# EPICS autosave request: xx_auto_transform_settings.req
$(P)$(T).DESC
$(P)$(T).SCAN
$(P)$(T).PREC
$(P)$(T).A
$(P)$(T).B
$(P)$(T).C
$(P)$(T).D
$(P)$(T).E
$(P)$(T).F
$(P)$(T).G
$(P)$(T).H
$(P)$(T).I
$(P)$(T).J
$(P)$(T).K
$(P)$(T).L
$(P)$(T).M
$(P)$(T).N
$(P)$(T).O
$(P)$(T).P
$(P)$(T).CMTA
$(P)$(T).CMTB
$(P)$(T).CMTC
$(P)$(T).CMTD
$(P)$(T).CMTE
$(P)$(T).CMTF
$(P)$(T).CMTG
$(P)$(T).CMTH
$(P)$(T).CMTI
$(P)$(T).CMTJ
$(P)$(T).CMTK
$(P)$(T).CMTL
$(P)$(T).CMTM
$(P)$(T).CMTN
$(P)$(T).CMTO
$(P)$(T).CMTP
$(P)$(T).CLCA
$(P)$(T).CLCB
$(P)$(T).CLCC
$(P)$(T).CLCD
$(P)$(T).CLCE
$(P)$(T).CLCF
$(P)$(T).CLCG
$(P)$(T).CLCH
$(P)$(T).CLCI
$(P)$(T).CLCJ
$(P)$(T).CLCK
$(P)$(T).CLCL
$(P)$(T).CLCM
$(P)$(T).CLCN
$(P)$(T).CLCO
$(P)$(T).CLCP
$(P)$(T).INPA
$(P)$(T).INPB
$(P)$(T).INPC
$(P)$(T).INPD
$(P)$(T).INPE
$(P)$(T).INPF
$(P)$(T).INPG
$(P)$(T).INPH
$(P)$(T).INPI
$(P)$(T).INPJ
$(P)$(T).INPK
$(P)$(T).INPL
$(P)$(T).INPM
$(P)$(T).INPN
$(P)$(T).INPO
$(P)$(T).INPP
$(P)$(T).OUTA
$(P)$(T).OUTB
$(P)$(T).OUTC
$(P)$(T).OUTD
$(P)$(T).OUTE
$(P)$(T).OUTF
$(P)$(T).OUTG
$(P)$(T).OUTH
$(P)$(T).OUTI
$(P)$(T).OUTJ
$(P)$(T).OUTK
$(P)$(T).OUTL
$(P)$(T).OUTM
$(P)$(T).OUTN
$(P)$(T).OUTO
$(P)$(T).OUTP
